// TIA Portal V16 export
// export: Created 2022-11-14T17:35:38.2779198Z, ExportSetting WithDefaults, DisplayName Totally Integrated Automation Portal, DisplayVersion V16, DisplayName TIA Portal Version Control Interface, DisplayVersion V16, DisplayName TIA Portal Openness, DisplayVersion V16, DisplayName STEP 7 Professional, DisplayVersion V16, DisplayName STEP 7 Safety, DisplayVersion V16, DisplayName WinCC Advanced, DisplayVersion V16
ORGANIZATION_BLOCK "Cyclic interrupt"   // OB30, LAD, CyclicInterrupt
TITLE = Rampa tiro
{ S7_Optimized_Access := 'TRUE' }
VERSION : 0.1
// Rampa per raggiungere tiro obiettivo e zero (0-20@100ms;20-100@20ms->3600ms)
// stored: AutoNumber true, IsIECCheckEnabled false, SetENOAutomatically false
   VAR_INPUT
      Initial_Call : Bool;   // Initial call of this OB
      Event_Count : Int;   // Events discarded
   END_VAR
   VAR_TEMP
      TempDint : DInt;
      TempDint_2 : DInt;
      TempInt : Int;
   END_VAR
   VAR_TEMP   // added for the SCL form of the ladder/FBD networks
      _w1 : Bool;
      _w2 : Bool;
   END_VAR
BEGIN

REGION Network 1: Impulso ogni 20ms (OB30)
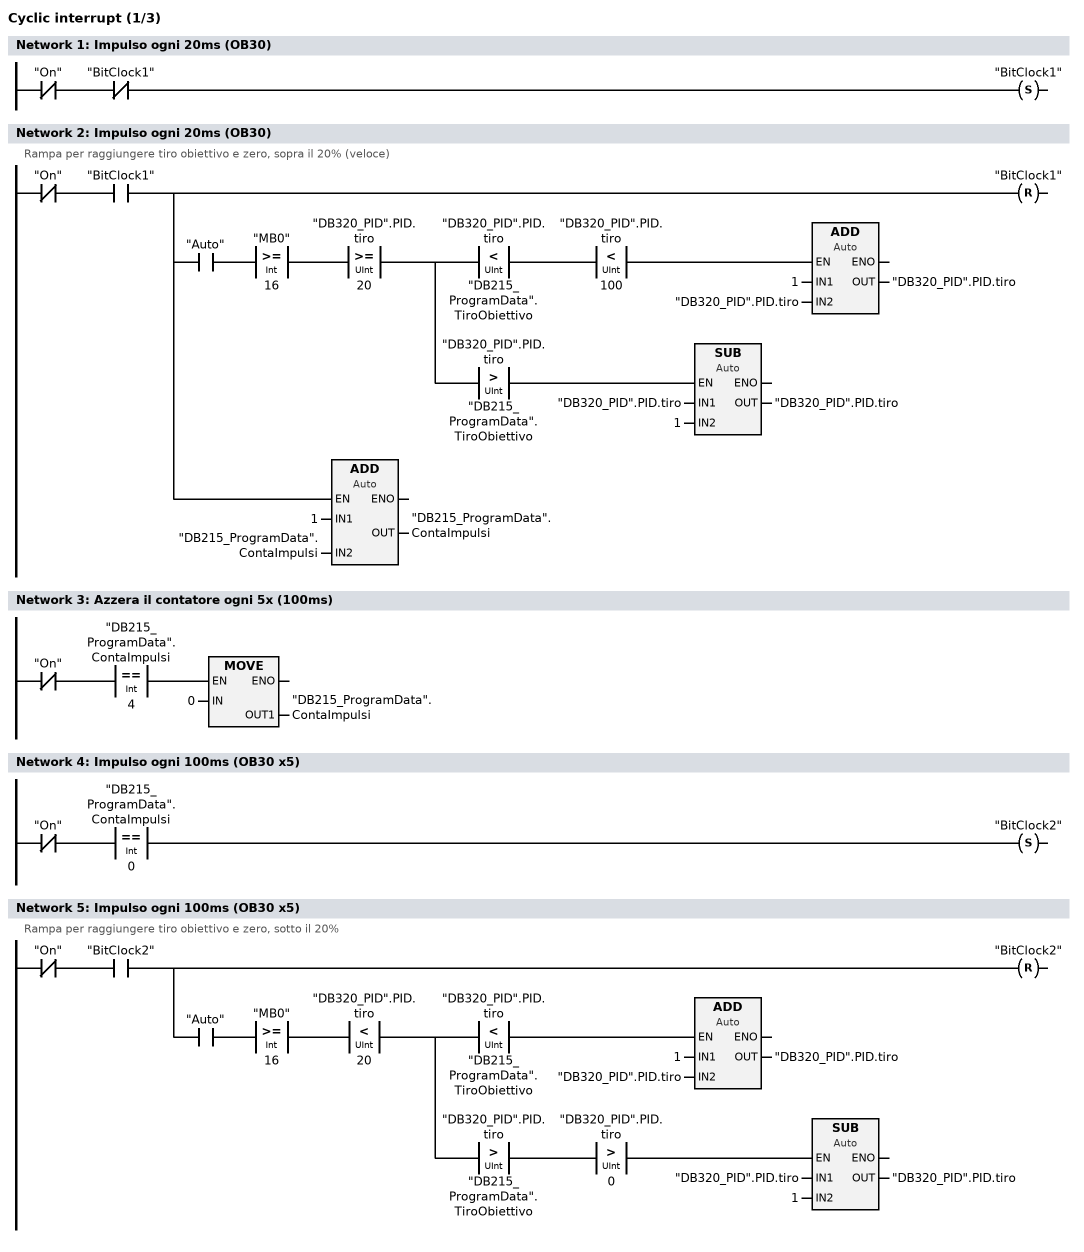
   RUNG wire#powerrail
      I_Contact( "On" )
      I_Contact( "BitClock1" )
      S_Coil( "BitClock1" )
   END_RUNG
   // the same network as SCL:
   IF NOT "On" AND NOT "BitClock1" THEN "BitClock1" := TRUE; END_IF;
END_REGION

REGION Network 2: Impulso ogni 20ms (OB30)
   // Rampa per raggiungere tiro obiettivo e zero, sopra il 20% (veloce)
   RUNG wire#powerrail
      I_Contact( "On" )
      Contact( "BitClock1" )
      wire#w1
      R_Coil( "BitClock1" )
   END_RUNG
   RUNG wire#w1
      Contact( "Auto" )
      { S7_Templates := "SrcType := Int" } GE_Contact(in1 := "MB0", in2 := 16)
      { S7_Templates := "SrcType := UInt" } GE_Contact(in1 := "DB320_PID".PID.tiro, in2 := 20)
      wire#w2
      { S7_Templates := "SrcType := UInt" } LT_Contact(in1 := "DB320_PID".PID.tiro, in2 := "DB215_ProgramData".TiroObiettivo)
      { S7_Templates := "SrcType := UInt" } LT_Contact(in1 := "DB320_PID".PID.tiro, in2 := 100)
      Add(in1 := 1, in2 := "DB320_PID".PID.tiro, out => "DB320_PID".PID.tiro)
   END_RUNG
   RUNG wire#w2
      { S7_Templates := "SrcType := UInt" } GT_Contact(in1 := "DB320_PID".PID.tiro, in2 := "DB215_ProgramData".TiroObiettivo)
      Sub(in1 := "DB320_PID".PID.tiro, in2 := 1, out => "DB320_PID".PID.tiro)
   END_RUNG
   RUNG wire#w1
      Add(in1 := 1, in2 := "DB215_ProgramData".ContaImpulsi, out => "DB215_ProgramData".ContaImpulsi)
   END_RUNG
   // the same network as SCL:
   #_w1 := NOT "On" AND "BitClock1";
   IF #_w1 THEN "BitClock1" := FALSE; END_IF;
   #_w2 := #_w1 AND "Auto" AND ("MB0" >= 16) AND ("DB320_PID".PID.tiro >= 20);
   IF #_w2 AND ("DB320_PID".PID.tiro < "DB215_ProgramData".TiroObiettivo) AND ("DB320_PID".PID.tiro < 100) THEN
       "DB320_PID".PID.tiro := 1 + "DB320_PID".PID.tiro;
   END_IF;
   IF #_w2 AND ("DB320_PID".PID.tiro > "DB215_ProgramData".TiroObiettivo) THEN
       "DB320_PID".PID.tiro := "DB320_PID".PID.tiro - 1;
   END_IF;
   IF #_w1 THEN "DB215_ProgramData".ContaImpulsi := 1 + "DB215_ProgramData".ContaImpulsi; END_IF;
END_REGION

REGION Network 3: Azzera il contatore ogni 5x (100ms)
   RUNG wire#powerrail
      I_Contact( "On" )
      { S7_Templates := "SrcType := Int" } EQ_Contact(in1 := "DB215_ProgramData".ContaImpulsi, in2 := 4)
      Move(in := 0, out1 => "DB215_ProgramData".ContaImpulsi)
   END_RUNG
   // the same network as SCL:
   IF NOT "On" AND ("DB215_ProgramData".ContaImpulsi = 4) THEN "DB215_ProgramData".ContaImpulsi := 0; END_IF;
END_REGION

REGION Network 4: Impulso ogni 100ms (OB30 x5)
   RUNG wire#powerrail
      I_Contact( "On" )
      { S7_Templates := "SrcType := Int" } EQ_Contact(in1 := "DB215_ProgramData".ContaImpulsi, in2 := 0)
      S_Coil( "BitClock2" )
   END_RUNG
   // the same network as SCL:
   IF NOT "On" AND ("DB215_ProgramData".ContaImpulsi = 0) THEN "BitClock2" := TRUE; END_IF;
END_REGION

REGION Network 5: Impulso ogni 100ms (OB30 x5)
   // Rampa per raggiungere tiro obiettivo e zero, sotto il 20%
   RUNG wire#powerrail
      I_Contact( "On" )
      Contact( "BitClock2" )
      wire#w1
      R_Coil( "BitClock2" )
   END_RUNG
   RUNG wire#w1
      Contact( "Auto" )
      { S7_Templates := "SrcType := Int" } GE_Contact(in1 := "MB0", in2 := 16)
      { S7_Templates := "SrcType := UInt" } LT_Contact(in1 := "DB320_PID".PID.tiro, in2 := 20)
      wire#w2
      { S7_Templates := "SrcType := UInt" } LT_Contact(in1 := "DB320_PID".PID.tiro, in2 := "DB215_ProgramData".TiroObiettivo)
      Add(in1 := 1, in2 := "DB320_PID".PID.tiro, out => "DB320_PID".PID.tiro)
   END_RUNG
   RUNG wire#w2
      { S7_Templates := "SrcType := UInt" } GT_Contact(in1 := "DB320_PID".PID.tiro, in2 := "DB215_ProgramData".TiroObiettivo)
      { S7_Templates := "SrcType := UInt" } GT_Contact(in1 := "DB320_PID".PID.tiro, in2 := 0)
      Sub(in1 := "DB320_PID".PID.tiro, in2 := 1, out => "DB320_PID".PID.tiro)
   END_RUNG
   // the same network as SCL:
   #_w1 := NOT "On" AND "BitClock2";
   IF #_w1 THEN "BitClock2" := FALSE; END_IF;
   #_w2 := #_w1 AND "Auto" AND ("MB0" >= 16) AND ("DB320_PID".PID.tiro < 20);
   IF #_w2 AND ("DB320_PID".PID.tiro < "DB215_ProgramData".TiroObiettivo) THEN
       "DB320_PID".PID.tiro := 1 + "DB320_PID".PID.tiro;
   END_IF;
   IF #_w2 AND ("DB320_PID".PID.tiro > "DB215_ProgramData".TiroObiettivo) AND ("DB320_PID".PID.tiro > 0) THEN
       "DB320_PID".PID.tiro := "DB320_PID".PID.tiro - 1;
   END_IF;
END_REGION

REGION Network 7: Arm rotation and top carriage speed change for DAC M20
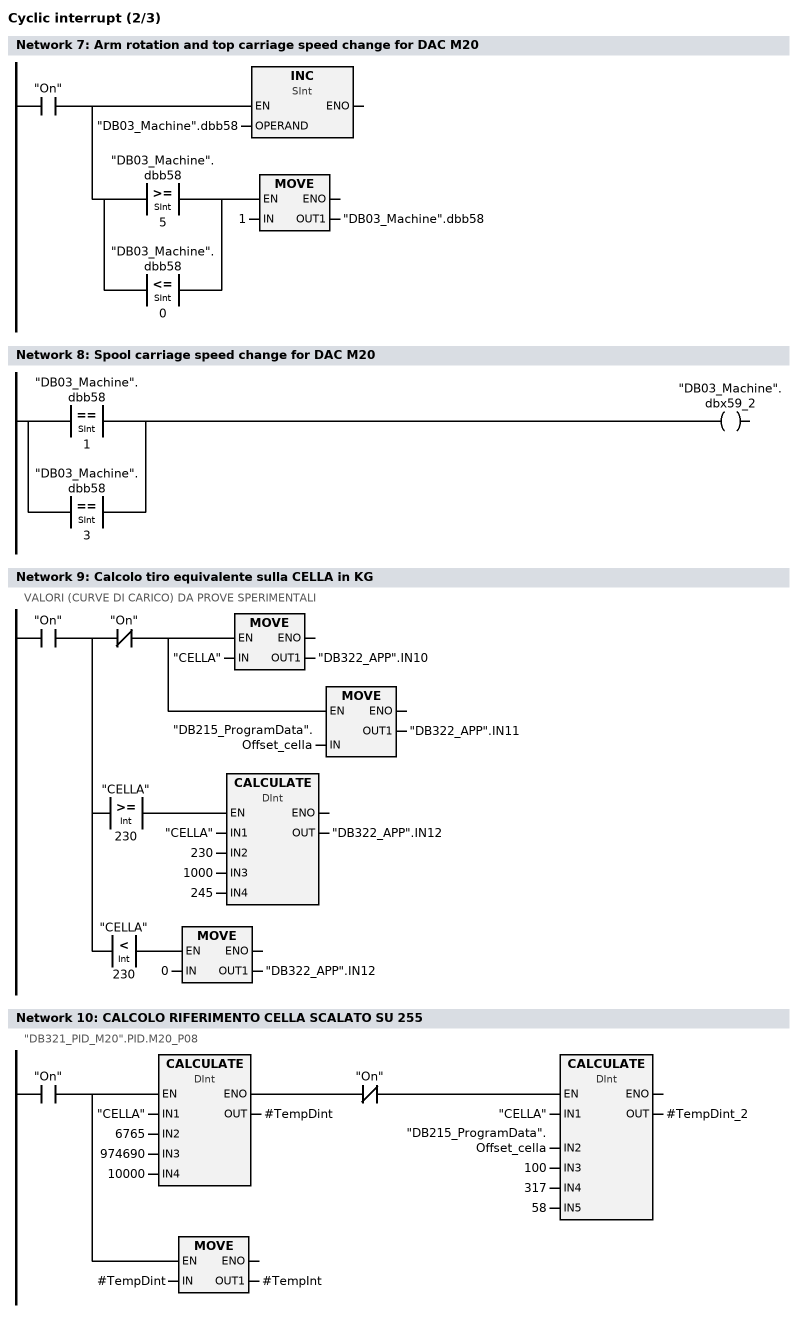
   RUNG wire#powerrail
      Contact( "On" )
      wire#w1
      { S7_Templates := "DestType := SInt"; S7_GenerateENO := "TRUE" } Inc( "DB03_Machine".dbb58 )
   END_RUNG
   RUNG wire#w1
      { S7_Templates := "SrcType := SInt" } GE_Contact(in1 := "DB03_Machine".dbb58, in2 := 5)
      wire#w2
      { S7_GenerateENO := "TRUE" } Move(in := 1, out1 => "DB03_Machine".dbb58)
   END_RUNG
   RUNG wire#w1
      { S7_Templates := "SrcType := SInt" } LE_Contact(in1 := "DB03_Machine".dbb58, in2 := 0)
   END_RUNG wire#w2
   // the same network as SCL:
   IF "On" THEN "DB03_Machine".dbb58 := "DB03_Machine".dbb58 + 1; END_IF;
   IF "On" AND (("DB03_Machine".dbb58 >= 5) OR ("DB03_Machine".dbb58 <= 0)) THEN
       "DB03_Machine".dbb58 := 1;
   END_IF;
END_REGION

REGION Network 8: Spool carriage speed change for DAC M20
   RUNG wire#powerrail
      { S7_Templates := "SrcType := SInt" } EQ_Contact(in1 := "DB03_Machine".dbb58, in2 := 1)
      wire#w1
      Coil( "DB03_Machine".dbx59_2 )
   END_RUNG
   RUNG wire#powerrail
      { S7_Templates := "SrcType := SInt" } EQ_Contact(in1 := "DB03_Machine".dbb58, in2 := 3)
   END_RUNG wire#w1
   // the same network as SCL:
   "DB03_Machine".dbx59_2 := ("DB03_Machine".dbb58 = 1) OR ("DB03_Machine".dbb58 = 3);
END_REGION

REGION Network 9: Calcolo tiro equivalente sulla CELLA in KG
   // VALORI (CURVE DI CARICO) DA PROVE SPERIMENTALI
   RUNG wire#powerrail
      Contact( "On" )
      wire#w1
      I_Contact( "On" )
      wire#w2
      Move(in := "CELLA", out1 => "DB322_APP".IN10)
   END_RUNG
   RUNG wire#w2
      Move(in := "DB215_ProgramData".Offset_cella, out1 => "DB322_APP".IN11)
   END_RUNG
   RUNG wire#w1
      { S7_Templates := "SrcType := Int" } GE_Contact(in1 := "CELLA", in2 := 230)
      { S7_Templates := "SrcType := DInt"; S7_Expression := "((IN1-IN2)*IN3)/IN4" } Calculate(in1 := "CELLA", in2 := 230, in3 := 1000, in4 := 245, out => "DB322_APP".IN12)
   END_RUNG
   RUNG wire#w1
      { S7_Templates := "SrcType := Int" } LT_Contact(in1 := "CELLA", in2 := 230)
      Move(in := 0, out1 => "DB322_APP".IN12)
   END_RUNG
   // the same network as SCL:
   IF "On" AND NOT "On" THEN
       "DB322_APP".IN10 := "CELLA";
       "DB322_APP".IN11 := "DB215_ProgramData".Offset_cella;
   END_IF;
   IF "On" AND ("CELLA" >= 230) THEN "DB322_APP".IN12 := (("CELLA"-230)*1000)/245; END_IF;
   IF "On" AND ("CELLA" < 230) THEN "DB322_APP".IN12 := 0; END_IF;
END_REGION

REGION Network 10: CALCOLO RIFERIMENTO CELLA SCALATO SU 255
   // "DB321_PID_M20".PID.M20_P08
   RUNG wire#powerrail
      Contact( "On" )
      wire#w1
      { S7_Templates := "SrcType := DInt"; S7_Expression := "(IN1*IN2-IN3)/IN4" } Calculate(in1 := "CELLA", in2 := 6765, in3 := 974690, in4 := 10000, out => #TempDint)
      I_Contact( "On" )
      { S7_Templates := "SrcType := DInt"; S7_Expression := "((IN1-IN2)*IN3/IN4)+IN5" } Calculate(in1 := "CELLA", in2 := "DB215_ProgramData".Offset_cella, in3 := 100, in4 := 317, in5 := 58, out => #TempDint_2)
   END_RUNG
   RUNG wire#w1
      Move(in := #TempDint, out1 => #TempInt)
   END_RUNG
   // the same network as SCL:
   IF "On" THEN #TempDint := ("CELLA"*6765-974690)/10000; END_IF;
   IF "On" AND NOT "On" THEN #TempDint_2 := (("CELLA"-"DB215_ProgramData".Offset_cella)*100/317)+58; END_IF;
   IF "On" THEN #TempInt := #TempDint; END_IF;
END_REGION

REGION Network 11: M20
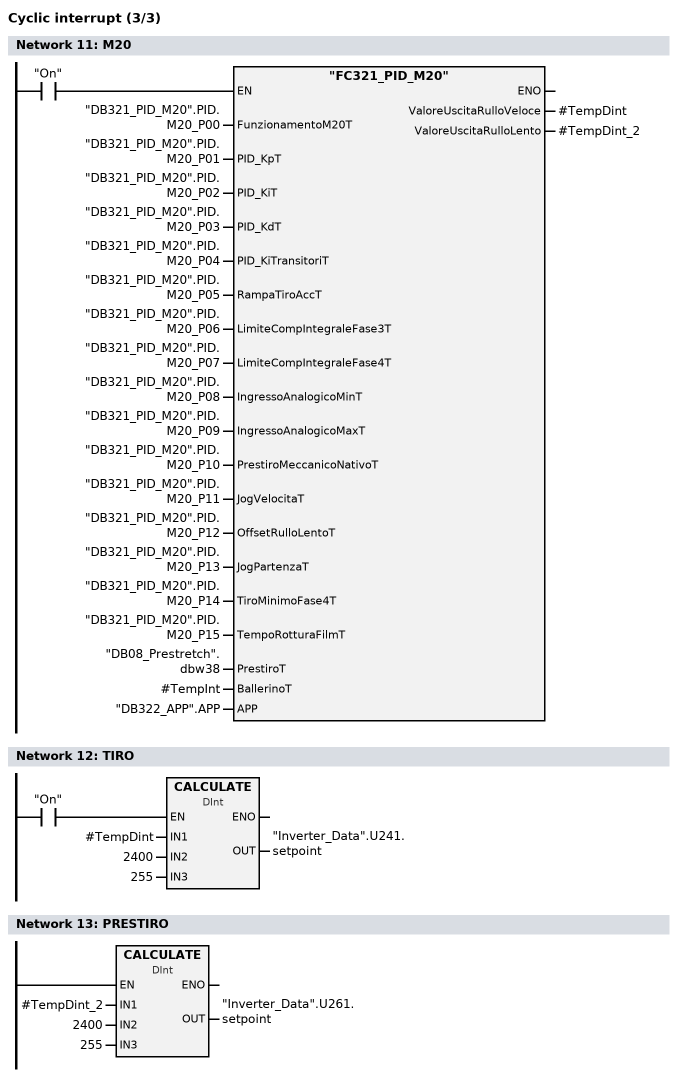
   RUNG wire#powerrail
      Contact( "On" )
      "FC321_PID_M20"(FunzionamentoM20T := "DB321_PID_M20".PID.M20_P00, PID_KpT := "DB321_PID_M20".PID.M20_P01, PID_KiT := "DB321_PID_M20".PID.M20_P02, PID_KdT := "DB321_PID_M20".PID.M20_P03, PID_KiTransitoriT := "DB321_PID_M20".PID.M20_P04, RampaTiroAccT := "DB321_PID_M20".PID.M20_P05, LimiteCompIntegraleFase3T := "DB321_PID_M20".PID.M20_P06, LimiteCompIntegraleFase4T := "DB321_PID_M20".PID.M20_P07, IngressoAnalogicoMinT := "DB321_PID_M20".PID.M20_P08, IngressoAnalogicoMaxT := "DB321_PID_M20".PID.M20_P09, PrestiroMeccanicoNativoT := "DB321_PID_M20".PID.M20_P10, JogVelocitaT := "DB321_PID_M20".PID.M20_P11, OffsetRulloLentoT := "DB321_PID_M20".PID.M20_P12, JogPartenzaT := "DB321_PID_M20".PID.M20_P13, TiroMinimoFase4T := "DB321_PID_M20".PID.M20_P14, TempoRotturaFilmT := "DB321_PID_M20".PID.M20_P15, PrestiroT := "DB08_Prestretch".dbw38, BallerinoT := #TempInt, APP := "DB322_APP".APP, ValoreUscitaRulloVeloce => #TempDint, ValoreUscitaRulloLento => #TempDint_2)
   END_RUNG
   // the same network as SCL:
   IF "On" THEN
       "FC321_PID_M20"(FunzionamentoM20T := "DB321_PID_M20".PID.M20_P00,
                       PID_KpT := "DB321_PID_M20".PID.M20_P01,
                       PID_KiT := "DB321_PID_M20".PID.M20_P02,
                       PID_KdT := "DB321_PID_M20".PID.M20_P03,
                       PID_KiTransitoriT := "DB321_PID_M20".PID.M20_P04,
                       RampaTiroAccT := "DB321_PID_M20".PID.M20_P05,
                       LimiteCompIntegraleFase3T := "DB321_PID_M20".PID.M20_P06,
                       LimiteCompIntegraleFase4T := "DB321_PID_M20".PID.M20_P07,
                       IngressoAnalogicoMinT := "DB321_PID_M20".PID.M20_P08,
                       IngressoAnalogicoMaxT := "DB321_PID_M20".PID.M20_P09,
                       PrestiroMeccanicoNativoT := "DB321_PID_M20".PID.M20_P10,
                       JogVelocitaT := "DB321_PID_M20".PID.M20_P11,
                       OffsetRulloLentoT := "DB321_PID_M20".PID.M20_P12,
                       JogPartenzaT := "DB321_PID_M20".PID.M20_P13,
                       TiroMinimoFase4T := "DB321_PID_M20".PID.M20_P14,
                       TempoRotturaFilmT := "DB321_PID_M20".PID.M20_P15,
                       PrestiroT := "DB08_Prestretch".dbw38,
                       BallerinoT := #TempInt,
                       APP := "DB322_APP".APP,
                       ValoreUscitaRulloVeloce => #TempDint,
                       ValoreUscitaRulloLento => #TempDint_2);
   END_IF;
END_REGION

REGION Network 12: TIRO
   RUNG wire#powerrail
      Contact( "On" )
      { S7_Templates := "SrcType := DInt"; S7_Expression := "IN1*IN2/IN3" } Calculate(in1 := #TempDint, in2 := 2400, in3 := 255, out => "Inverter_Data".U241.setpoint)
   END_RUNG
   // the same network as SCL:
   IF "On" THEN "Inverter_Data".U241.setpoint := #TempDint*2400/255; END_IF;
END_REGION

REGION Network 13: PRESTIRO
   RUNG wire#powerrail
      { S7_Templates := "SrcType := DInt"; S7_Expression := "IN1*IN2/IN3" } Calculate(in1 := #TempDint_2, in2 := 2400, in3 := 255, out => "Inverter_Data".U261.setpoint)
   END_RUNG
   // the same network as SCL:
   "Inverter_Data".U261.setpoint := #TempDint_2*2400/255;
END_REGION
END_ORGANIZATION_BLOCK
